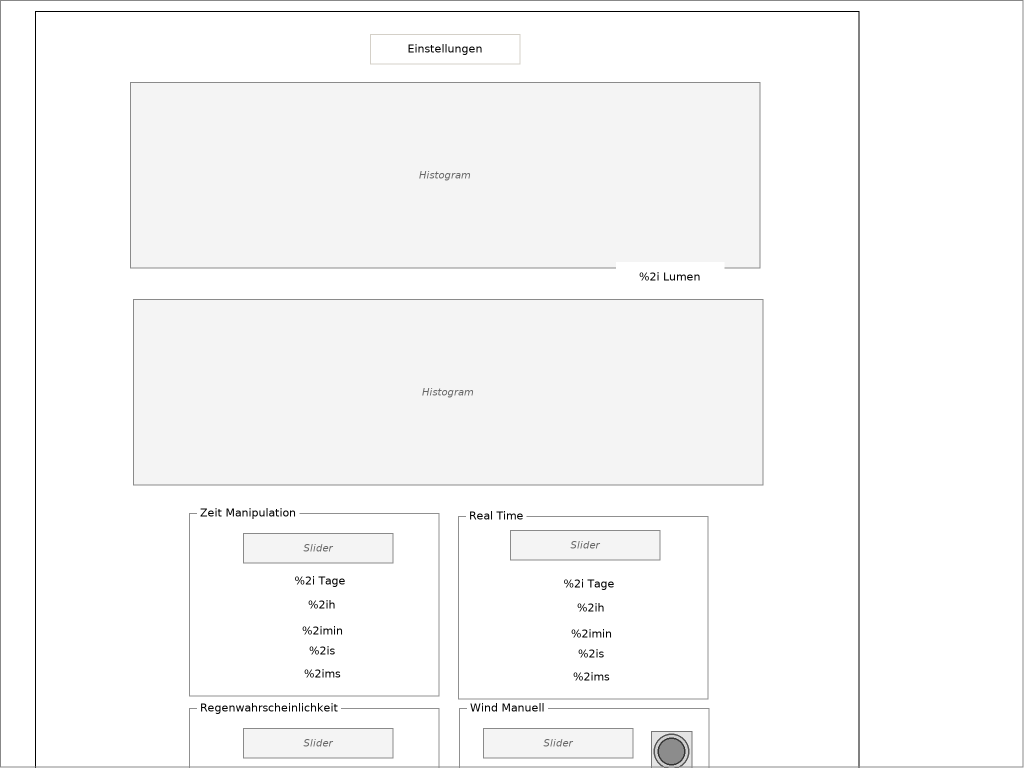
VISUALIZATION Settings  // 1024x768
    Rectangle (35,11 824x973)
    Histogram (130,82 630x186), scale format: %i, scale 0..3000
        p1518820177: SonneHistory
        p102497268: SonneHistory
        p788070771: ARRAY [0..DatenHistoryZaehler] OF INT
    GroupBox (189,505 250x191), "Zeit Manipulation"
        Slider (54,28 150x30), variable: SimZeitMultiplikator, scale 0..4
        Textfield (102,61 62x30), "%2i Tage", text variable: SimRealTagSeitStart
        Textfield (101,111 65x30), "%2imin", text variable: SimMinute
        Textfield (100,131 66x30), "%2is", text variable: SimSekunde
        Textfield (100,154 67x30), "%2ims", text variable: SimMilliSekunde
        Textfield (102,85 62x30), "%2ih", text variable: SimStunde
    GroupBox (458,508 250x191), "Real Time"
        Textfield (102,61 62x30), "%2i Tage", text variable: RealTagSeitStart
        Slider (52,22 150x30), variable: RealtimeManipulator, scale 0..3
        Textfield (101,111 65x30), "%2imin", text variable: RealMinute
        Textfield (100,131 66x30), "%2is", text variable: RealSekunde
        Textfield (100,154 67x30), "%2ims", text variable: RealMilliSekunde
        Textfield (102,85 62x30), "%2ih", text variable: RealStunde
    Textfield (616,262 108x30), "%2i Lumen", text variable: Licht
    GroupBox (189,700 250x105), "Regenwahrscheinlichkeit"
        Slider (54,28 150x30), variable: Regenwahrscheinlichkeit, scale 0..100
        Textfield (32,61 205x30), "%i %", text variable: Regenwahrscheinlichkeit
    Textfield (370,34 150x30), "Einstellungen"
    Button (680,929 150x30), "Schliessen"
        OnMouseClick: CloseDialog Dialog=Settings, Result=OK, NumpadKeypadSet=True
    Histogram (133,299 630x186), scale format: %i, scale 0..500
        p1518820177: WindHistory
        p102497268: WindHistory
        p788070771: ARRAY [0..DatenHistoryZaehler] OF REAL
    GroupBox (459,700 250x105), "Wind Manuell"
        Slider (24,28 150x30), variable: Wind_V, scale 0..200
        Textfield (2,61 205x30), "%i km/h Wind", text variable: net_wind
        PushSwitch (192,31 41x41), variable: Wind_Auto_V, behaviour: TAP, style: Switch-PushSwitch-Gray
    GroupBox (189,816 250x105), "Sonne Manuell"
        Slider (40,28 150x30), variable: Sonne_V, scale 100..2500
        Textfield (44,65 139x30), "%i Lumen", text variable: net_sonne
        PushSwitch (197,32 41x41), variable: Sonne_Auto_V, behaviour: TAP, style: Switch-PushSwitch-Gray
    PushSwitch (486,830 41x41), variable: GL_Besucher_reset, behaviour: TAP, style: Switch-PushSwitch-Gray
    PushSwitch (486,878 43x45), variable: GL_Alarm_reset, behaviour: TAP, style: Switch-PushSwitch-Gray
    Textfield (543,838 213x23), "Besucher zurücksetzen"
    Textfield (541,881 196x30), "Alarm zurücksetzen"
END_VISUALIZATION

(* stored: Version 1.1.0.1, ProductVersion 3.1.4018.5
   Visu Settings: Id {0236438a-636b-48a4-bb82-1f0497612fc4} *)
